Staubli VAL3: Home.pjx

--- Home.pjx ---
Parameters version=s7.8.3 stackSize=5000 millimeterUnit=true
Program file=Edit.pgx
Program file=EnterPageKey.pgx
Program file=Main.pgx
Program file=MainKey.pgx
Program file=OnF1.pgx
Program file=OnF2.pgx
Program file=OnF7.pgx
Program file=OnF8.pgx
Program file=Refresh.pgx
Program file=RefreshList.pgx
Program file=start.pgx
Program file=stop.pgx
Data file=Home.dtx
Library alias=user path=Disk://userPage/USERPAGE.pjx
Library alias=PublicData path=Disk://PublicData/PublicData.pjx

--- Home.dtx ---
mdesc mNomSpeed
bool bUserRefresh
bool bListRefresh
num nSelected
string sItem
bool bExit
string sParameter
string sListItemValue
string sList
num nType
mdesc mHome = {accel=10, decel=10, tmax=100, leave=1, reach=1, blend=cartesian}

--- Main.pgx ---
public program Main()
  local num l_nKey
begin
  //
  bUserRefresh=bListRefresh=true
  bExit=false
  //
  do
    call Refresh()
    call RefreshList()
    call user:setList("",sList,bUserRefresh,bListRefresh,nSelected,sItem,l_nKey)
    bUserRefresh=false
    bListRefresh=false
    call MainKey(l_nKey)
    delay(0)
  until bExit

end

--- start.pgx ---
public program start()
begin
  //
  call Edit()
end

--- Edit.pgx ---
program Edit()
  local bool l_bRes
  local num l_i
  local string l_sValue
  local num l_nSelect
  local string l_sItem
  local num l_nKey
  local num l_nRes
begin

  cls()
  resize(sParameter,1,6)
  sParameter[0]="j1"
  sParameter[1]="j2"
  sParameter[2]="j3"
  sParameter[3]="j4"
  sParameter[4]="j5"
  sParameter[5]="j6"
  //
  resize(sListItemValue,1,size(sParameter))
  sListItemValue[0]=toString(".3",PublicData:jHome.j1)
  sListItemValue[1]=toString(".3",PublicData:jHome.j2)
  sListItemValue[2]=toString(".3",PublicData:jHome.j3)
  sListItemValue[3]=toString(".3",PublicData:jHome.j4)
  sListItemValue[4]=toString(".3",PublicData:jHome.j5)
  sListItemValue[5]=toString(".3",PublicData:jHome.j6)
  //
  for l_i=0 to size(sParameter)-1
    call user:strlength(sParameter[l_i],user:nBottomX/2)
    l_sValue=sListItemValue[l_i]
    call user:strlength(l_sValue,user:nBottomX/2+1)
    sParameter[l_i]=sParameter[l_i]+":"+l_sValue
  endFor

  bUserRefresh=true
  bListRefresh=true
  //
  do
    if bUserRefresh
      cls()
      userPage()
      gotoxy(1,1)
      put("F1->记录")
      call user:clear(0,13)
      gotoxy(1,13)
      put("F1")
      gotoxy(1,2)
      put("F2->移动")
      gotoxy(6,13)
      put("F2")
      call user:typeMenu(8,"确定")
    endIf
    call user:setList(sItem,sParameter,bUserRefresh,bListRefresh,l_nSelect,l_sItem,l_nKey)
    bUserRefresh=false
    bListRefresh=false
    call EnterPageKey(l_nKey,l_nSelect,sParameter[l_nSelect])
    delay(0)
  until l_nKey==255 or l_nKey==278
  if l_nKey==278
    PublicData:libSave()
  endIf
  bUserRefresh=true
  bListRefresh=true
end

--- EnterPageKey.pgx ---
program EnterPageKey(num& x_nKey, num& x_nSelect, string& x_sItem)
  local string l_sStr
  local num l_nKey
  local string l_sEmpty
  local string l_sValue
  local num l_nItem
  local num l_nView
  local string l_sItem
  local point lp
  local string l_sYN[2]
  local bool l_bRes
  local num l_i
  local num l_nWorkMode
  local num l_nStatus
begin
  //
  switch x_nSelect
    case 0
      if x_nKey==270
        call user:editNum(x_sItem,sListItemValue[x_nSelect],PublicData:jHome.j1,x_nSelect)
      endIf
    break
    case 1
      if x_nKey==270
        call user:editNum(x_sItem,sListItemValue[x_nSelect],PublicData:jHome.j2,x_nSelect)
      endIf
    break
    case 2
      if x_nKey==270
        call user:editNum(x_sItem,sListItemValue[x_nSelect],PublicData:jHome.j3,x_nSelect)
      endIf
    break
    case 3
      if x_nKey==270
        call user:editNum(x_sItem,sListItemValue[x_nSelect],PublicData:jHome.j4,x_nSelect)
      endIf
    break
    case 4
      if x_nKey==27
        call user:editNum(x_sItem,sListItemValue[x_nSelect],PublicData:jHome.j5,x_nSelect)
      endIf
    break
    case 5
      if x_nKey==270
        call user:editNum(x_sItem,sListItemValue[x_nSelect],PublicData:jHome.j6,x_nSelect)
      endIf
    break
  endSwitch
  if x_nKey==271
    PublicData:jHome=herej()
    sParameter[0]="j1"
    sParameter[1]="j2"
    sParameter[2]="j3"
    sParameter[3]="j4"
    sParameter[4]="j5"
    sParameter[5]="j6"
    sListItemValue[0]=toString(".3",PublicData:jHome.j1)
    sListItemValue[1]=toString(".3",PublicData:jHome.j2)
    sListItemValue[2]=toString(".3",PublicData:jHome.j3)
    sListItemValue[3]=toString(".3",PublicData:jHome.j4)
    sListItemValue[4]=toString(".3",PublicData:jHome.j5)
    sListItemValue[5]=toString(".3",PublicData:jHome.j6)
    for l_i=0 to size(sParameter)-1
      call user:strlength(sParameter[l_i],user:nBottomX/2)
      l_sValue=sListItemValue[l_i]
      call user:strlength(l_sValue,user:nBottomX/2+1)
      sParameter[l_i]=sParameter[l_i]+":"+l_sValue
    endFor
    popUpMsg("记录完成")
  endIf

  if x_nKey==272
    l_nWorkMode=workingMode(l_nStatus)
    if l_nWorkMode!=1
      popUpMsg("切换到手动模式")
      return
    endIf
    call user:timerDialog("正在回安全点......",0)
      movej(PublicData:jHome,flange,mHome)
      waitEndMove()
    endIf


  if x_nKey==270 or x_nKey==271 or x_nKey==272
    bUserRefresh=true
    bListRefresh=true
  endIf
end

--- MainKey.pgx ---
program MainKey(num x_nKey)
  local num l_nKey
begin
  //
  switch x_nKey
    //
    case 271
      call OnF1()
    break
    //编辑
    case 272
      call OnF2()
    break
    //
    case 273
      //call OnF3()
    break
    //
    case 274
     // call OnF4()
    break
    //
    case 275
    break
    //
    case 276
      //call OnF6()
    break
    //save
    case 277
      call OnF7()
    break
    //返回
    case 278
      call OnF8("是否返回")
    break

  endSwitch
end

--- OnF1.pgx ---
program OnF1()
begin

end

--- OnF7.pgx ---
program OnF7()
begin
  //
  libSave()
  popUpMsg("保存完毕!")
end

--- Refresh.pgx ---
program Refresh()
begin
  //
//  if bUserRefresh
////    cls()
//    userPage()
//    if nType==1
//      gotoxy(1,1)
//      put("F1->确定")
//      gotoxy(1,13)
//      put("F1")
//    endIf

//    gotoxy(1,2)
//    put("F2->编辑")
//    gotoxy(6,13)
//    put("F2")
//    //    gotoxy(1,3)
//    //    put("F3->删除")
//    //    gotoxy(11,13)
//    //    put("F3")
//    //    gotoxy(1,4)
//    //    put("F4->编辑路径")
//    //    gotoxy(16,13)
//    //    put("编辑")
//    //
//    //    gotoxy(1,6)
//    //    put("F6->")
//    //    gotoxy(26,13)
//    //    put("")
//    gotoxy(1,7)
//    put("F7->保存")
//    gotoxy(31,13)
//    put("F7")
//    gotoxy(1,8)
//    put("F8->返回")
//    gotoxy(36,13)
//    put("F8")
//  endIf
end

--- RefreshList.pgx ---
program RefreshList()
  local num l_ni
begin
  //
  if bListRefresh
    sParameter[0]="j1"
    sParameter[1]="j2"
    sParameter[2]="j3"
    sParameter[3]="j4"
    sParameter[4]="j5"
    sParameter[5]="j6"
    //
    sListItemValue[0]=toString(".3",PublicData:jHome.j1)
    sListItemValue[1]=toString(".3",PublicData:jHome.j2)
    sListItemValue[2]=toString(".3",PublicData:jHome.j3)
    sListItemValue[3]=toString(".3",PublicData:jHome.j4)
    sListItemValue[4]=toString(".3",PublicData:jHome.j5)
    sListItemValue[5]=toString(".3",PublicData:jHome.j6)
  endIf

end
